Staubli VAL3: GetAxisStatus.pgx

public program GetAxisStatus(bool& x_bBPower (dimensions=1), bool& x_nAlarm (dimensions=1), bool& x_nBackHome (dimensions=1))
begin
  x_bBPower=(dDio["In4_b7MotorPower"]==true)
  x_nAlarm=(dDio["In4_b7MotorError"]==true)
  x_nBackHome=(dDio["In4_b7BackHome"]==true)
end
